Staubli VAL3: readDataOnce.pgx

program readDataOnce(sio& x_UdpSocket, num& x_nData[], bool& x_bNewData, bool& x_bError)
  local num l_nSioReadBytes
begin
  x_bNewData = false
  x_bError = false

  // Read from UDP socket
  l_nSioReadBytes = sioGet(x_UdpSocket, x_nData)

  if(l_nSioReadBytes == size(x_nData))
    // Successfully read a full message
    x_bNewData = true
  elseIf (l_nSioReadBytes > 0)
    // Message of wrong size received, error
    logMsg("ros2_server::readDataOnce : message of wrong size received", 2)
    x_bError = true
    return
  endIf
end
